Yaskawa INFORM job: kufsa_angle.JBI

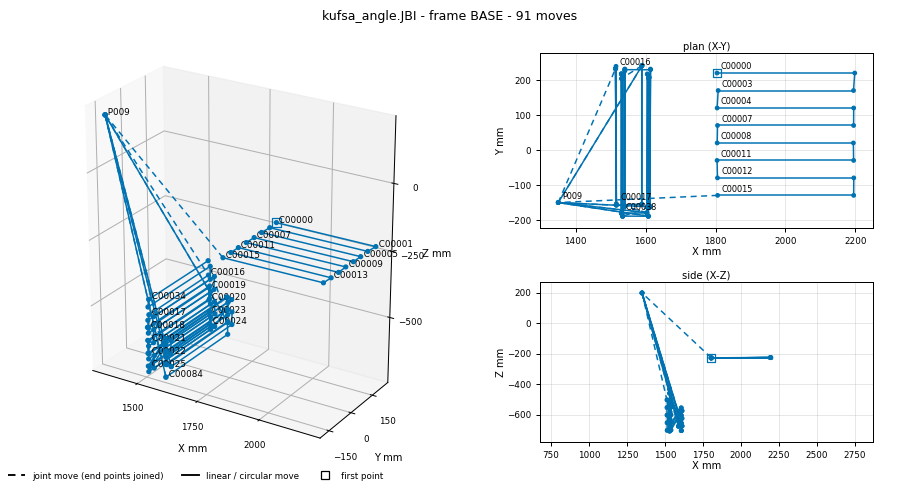
[picture p0: tool path of kufsa_angle.JBI in frame BASE, 91 of 91 moves have a stored position in this frame; points joined in program order, loops and branches not executed]
/JOB
//NAME kufsa_angle
//POS
///NPOS 86,0,86,1,0,0
///TOOL 0
///POSTYPE BASE
///RECTAN
///RCONF 0,0,0,0,0,0,0,0,0,0,0,0,0,0,0,0,0,0,0,0,0,0,0,0
C00000=1804.266,220.599,-227.332,179.0000,1.0000,1.0000
C00001=2198.370,220.599,-225.837,179.0000,1.0000,1.0000
C00002=2194.801,170.599,-225.649,179.0000,1.0000,1.0000
C00003=1807.577,170.599,-227.559,179.0000,1.0000,1.0000
C00004=1804.622,120.599,-227.769,179.0000,1.0000,1.0000
C00005=2195.335,120.599,-225.843,179.0000,1.0000,1.0000
C00006=2195.106,70.599,-225.320,179.0000,1.0000,1.0000
C00007=1805.716,70.599,-228.029,179.0000,1.0000,1.0000
C00008=1804.735,20.599,-228.045,179.0000,1.0000,1.0000
C00009=2194.418,20.599,-225.391,179.0000,1.0000,1.0000
C00010=2195.097,-29.400,-225.681,179.0000,1.0000,1.0000
C00011=1804.440,-29.400,-228.141,179.0000,1.0000,1.0000
C00012=1805.619,-79.400,-227.256,179.0000,1.0000,1.0000
C00013=2195.630,-79.400,-225.700,179.0000,1.0000,1.0000
C00014=2195.292,-129.400,-224.241,179.0000,1.0000,1.0000
C00015=1805.953,-129.400,-227.208,179.0000,1.0000,1.0000
C00016=1513.631,232.354,-503.993,179.0000,-89.9999,1.0000
C00017=1516.149,-153.231,-503.993,179.0000,-89.9999,1.0000
C00018=1516.042,-157.471,-553.993,179.0000,-89.9999,1.0000
C00019=1513.923,233.133,-553.993,179.0000,-89.9999,1.0000
C00020=1514.033,233.523,-603.993,179.0000,-89.9999,1.0000
C00021=1516.196,-156.884,-603.993,179.0000,-89.9999,1.0000
C00022=1516.145,-156.999,-653.993,179.0000,-89.9999,1.0000
C00023=1514.649,233.710,-653.993,179.0000,-89.9999,1.0000
C00024=1515.282,239.938,-703.993,179.0000,-89.9999,1.0000
C00025=1516.324,-157.007,-703.993,179.0000,-89.9999,1.0000
C00026=1588.761,-154.348,-577.217,180.0000,-45.0000,0.0000
C00027=1588.933,240.643,-577.217,180.0000,-45.0000,0.0000
C00028=1588.993,242.129,-627.217,180.0000,-45.0000,0.0000
C00029=1589.153,-155.140,-627.217,180.0000,-45.0000,0.0000
C00030=1589.056,-155.290,-677.217,180.0000,-45.0000,0.0000
C00031=1589.812,241.960,-677.217,180.0000,-45.0000,0.0000
C00032=1589.812,241.960,-677.217,180.0000,-45.0000,0.0000
C00033=1530.443,204.779,-432.522,179.0000,-89.9999,1.0000
C00034=1531.499,-175.214,-432.522,179.0000,-89.9999,1.0000
C00035=1531.405,-179.918,-459.727,179.0000,-89.9999,1.0000
C00036=1530.485,218.119,-459.727,179.0000,-89.9999,1.0000
C00037=1531.882,216.269,-509.727,179.0000,-89.9999,1.0000
C00038=1531.275,-181.949,-509.727,179.0000,-89.9999,1.0000
C00039=1531.305,-180.389,-559.727,179.0000,-89.9999,1.0000
C00040=1531.688,217.320,-559.727,179.0000,-89.9999,1.0000
C00041=1530.439,218.736,-609.727,179.0000,-89.9999,1.0000
C00042=1531.606,-180.718,-609.727,179.0000,-89.9999,1.0000
C00043=1530.852,-180.562,-659.727,179.0000,-89.9999,1.0000
C00044=1531.645,217.737,-659.727,179.0000,-89.9999,1.0000
C00045=1532.334,216.222,-709.727,179.0000,-89.9999,1.0000
C00046=1530.209,-180.083,-709.727,179.0000,-89.9999,1.0000
C00047=1603.447,-179.797,-582.950,180.0000,-45.0000,0.0000
C00048=1605.418,217.726,-582.950,180.0000,-45.0000,0.0000
C00049=1604.594,217.605,-632.950,180.0000,-45.0000,0.0000
C00050=1603.382,-179.006,-632.950,180.0000,-45.0000,0.0000
C00051=1603.382,-179.006,-632.950,180.0000,-45.0000,0.0000
C00052=1540.494,-160.372,-502.282,179.0000,-89.9999,1.0000
C00053=1540.352,230.020,-502.282,179.0000,-89.9999,1.0000
C00054=1540.533,226.582,-552.282,179.0000,-89.9999,1.0000
C00055=1540.232,-160.082,-552.282,179.0000,-89.9999,1.0000
C00056=1539.904,-161.733,-602.282,179.0000,-89.9999,1.0000
C00057=1540.218,229.622,-602.282,179.0000,-89.9999,1.0000
C00058=1540.573,232.252,-652.282,179.0000,-89.9999,1.0000
C00059=1540.340,-160.160,-652.282,179.0000,-89.9999,1.0000
C00060=1539.291,-159.918,-702.282,179.0000,-89.9999,1.0000
C00061=1540.509,230.302,-702.282,179.0000,-89.9999,1.0000
C00062=1613.808,230.041,-575.506,180.0000,-45.0000,0.0000
C00063=1612.459,-160.195,-575.506,180.0000,-45.0000,0.0000
C00064=1611.652,-164.339,-625.506,180.0000,-45.0000,0.0000
C00065=1613.824,231.968,-625.506,180.0000,-45.0000,0.0000
C00066=1613.735,230.903,-675.506,180.0000,-45.0000,0.0000
C00067=1612.429,-162.123,-675.506,180.0000,-45.0000,0.0000
C00068=1612.429,-162.123,-675.506,180.0000,-45.0000,0.0000
C00069=1534.042,-189.208,-533.001,179.0000,-89.9999,1.0000
C00070=1534.110,208.321,-533.001,179.0000,-89.9999,1.0000
C00071=1533.962,207.490,-583.001,179.0000,-89.9999,1.0000
C00072=1534.342,-189.439,-583.001,179.0000,-89.9999,1.0000
C00073=1534.609,-189.394,-633.001,179.0000,-89.9999,1.0000
C00074=1534.722,207.440,-633.001,179.0000,-89.9999,1.0000
C00075=1535.013,204.575,-683.001,179.0000,-89.9999,1.0000
C00076=1534.488,-188.796,-683.001,179.0000,-89.9999,1.0000
C00077=1607.894,-189.015,-556.224,180.0000,-45.0000,0.0000
C00078=1608.406,204.586,-556.224,180.0000,-45.0000,0.0000
C00079=1609.291,208.155,-606.224,180.0000,-45.0000,0.0000
C00080=1607.577,-189.129,-606.224,180.0000,-45.0000,0.0000
C00081=1607.618,-188.869,-656.224,180.0000,-45.0000,0.0000
C00082=1609.664,207.585,-656.224,180.0000,-45.0000,0.0000
C00083=1610.137,208.269,-706.224,180.0000,-45.0000,0.0000
C00084=1607.691,-188.817,-706.224,180.0000,-45.0000,0.0000
C00085=1607.691,-188.817,-706.224,180.0000,-45.0000,0.0000
///POSTYPE PULSE
///PULSE
EC00000=0
EC00001=0
EC00002=0
EC00003=0
EC00004=0
EC00005=0
EC00006=0
EC00007=0
EC00008=0
EC00009=0
EC00010=0
EC00011=0
EC00012=0
EC00013=0
EC00014=0
EC00015=0
EC00016=0
EC00017=0
EC00018=0
EC00019=0
EC00020=0
EC00021=0
EC00022=0
EC00023=0
EC00024=0
EC00025=0
EC00026=0
EC00027=0
EC00028=0
EC00029=0
EC00030=0
EC00031=0
EC00032=92160
EC00033=92160
EC00034=92160
EC00035=92160
EC00036=92160
EC00037=92160
EC00038=92160
EC00039=92160
EC00040=92160
EC00041=92160
EC00042=92160
EC00043=92160
EC00044=92160
EC00045=92160
EC00046=92160
EC00047=92160
EC00048=92160
EC00049=92160
EC00050=92160
EC00051=184320
EC00052=184320
EC00053=184320
EC00054=184320
EC00055=184320
EC00056=184320
EC00057=184320
EC00058=184320
EC00059=184320
EC00060=184320
EC00061=184320
EC00062=184320
EC00063=184320
EC00064=184320
EC00065=184320
EC00066=184320
EC00067=184320
EC00068=276480
EC00069=276480
EC00070=276480
EC00071=276480
EC00072=276480
EC00073=276480
EC00074=276480
EC00075=276480
EC00076=276480
EC00077=276480
EC00078=276480
EC00079=276480
EC00080=276480
EC00081=276480
EC00082=276480
EC00083=276480
EC00084=276480
EC00085=368640
///POSTYPE BASE
///RECTAN
///RCONF 1,0,0,0,0,0,0,0,0,0,0,0,0,0,0,0,0,0,0,0,0,0,0,0
P00009=1350.000,-150.000,200.000,-180.0000,-45.0000,0.0000
//INST
///DATE 2023/01/18 16:57
///ATTR SC,RW,RJ
////FRAME BASE
///GROUP1 RB1,ST1
NOP
MOVJ C00000 EC00000 VJ=15.00
CALL JOB:SPYON
MOVL C00001 EC00001 V=200.0
MOVL C00002 EC00002 V=200.0
MOVL C00003 EC00003 V=200.0
MOVL C00004 EC00004 V=200.0
MOVL C00005 EC00005 V=200.0
MOVL C00006 EC00006 V=200.0
MOVL C00007 EC00007 V=200.0
MOVL C00008 EC00008 V=200.0
MOVL C00009 EC00009 V=200.0
MOVL C00010 EC00010 V=200.0
MOVL C00011 EC00011 V=200.0
MOVL C00012 EC00012 V=200.0
MOVL C00013 EC00013 V=200.0
MOVL C00014 EC00014 V=200.0
MOVL C00015 EC00015 V=200.0
CALL JOB:SPYOF
MOVJ P009 VJ=15.00
MOVJ C00016 EC00016 VJ=15.00
CALL JOB:SPYON
MOVL C00017 EC00017 V=200.0
MOVL C00018 EC00018 V=200.0
MOVL C00019 EC00019 V=200.0
MOVL C00020 EC00020 V=200.0
MOVL C00021 EC00021 V=200.0
MOVL C00022 EC00022 V=200.0
MOVL C00023 EC00023 V=200.0
MOVL C00024 EC00024 V=200.0
MOVL C00025 EC00025 V=200.0
MOVL C00026 EC00026 V=200.0
MOVL C00027 EC00027 V=200.0
MOVL C00028 EC00028 V=200.0
MOVL C00029 EC00029 V=200.0
MOVL C00030 EC00030 V=200.0
MOVL C00031 EC00031 V=200.0
CALL JOB:SPYOF
MOVJ P009 VJ=15.00
MOVL C00032 EC00032 V=200.0
MOVJ C00033 EC00033 VJ=15.00
CALL JOB:SPYON
MOVL C00034 EC00034 V=200.0
MOVL C00035 EC00035 V=200.0
MOVL C00036 EC00036 V=200.0
MOVL C00037 EC00037 V=200.0
MOVL C00038 EC00038 V=200.0
MOVL C00039 EC00039 V=200.0
MOVL C00040 EC00040 V=200.0
MOVL C00041 EC00041 V=200.0
MOVL C00042 EC00042 V=200.0
MOVL C00043 EC00043 V=200.0
MOVL C00044 EC00044 V=200.0
MOVL C00045 EC00045 V=200.0
MOVL C00046 EC00046 V=200.0
MOVL C00047 EC00047 V=200.0
MOVL C00048 EC00048 V=200.0
MOVL C00049 EC00049 V=200.0
MOVL C00050 EC00050 V=200.0
CALL JOB:SPYOF
MOVJ P009 VJ=15.00
MOVL C00051 EC00051 V=200.0
MOVJ C00052 EC00052 VJ=15.00
CALL JOB:SPYON
MOVL C00053 EC00053 V=200.0
MOVL C00054 EC00054 V=200.0
MOVL C00055 EC00055 V=200.0
MOVL C00056 EC00056 V=200.0
MOVL C00057 EC00057 V=200.0
MOVL C00058 EC00058 V=200.0
MOVL C00059 EC00059 V=200.0
MOVL C00060 EC00060 V=200.0
MOVL C00061 EC00061 V=200.0
MOVL C00062 EC00062 V=200.0
MOVL C00063 EC00063 V=200.0
MOVL C00064 EC00064 V=200.0
MOVL C00065 EC00065 V=200.0
MOVL C00066 EC00066 V=200.0
MOVL C00067 EC00067 V=200.0
CALL JOB:SPYOF
MOVJ P009 VJ=15.00
MOVL C00068 EC00068 V=200.0
MOVJ C00069 EC00069 VJ=15.00
CALL JOB:SPYON
MOVL C00070 EC00070 V=200.0
MOVL C00071 EC00071 V=200.0
MOVL C00072 EC00072 V=200.0
MOVL C00073 EC00073 V=200.0
MOVL C00074 EC00074 V=200.0
MOVL C00075 EC00075 V=200.0
MOVL C00076 EC00076 V=200.0
MOVL C00077 EC00077 V=200.0
MOVL C00078 EC00078 V=200.0
MOVL C00079 EC00079 V=200.0
MOVL C00080 EC00080 V=200.0
MOVL C00081 EC00081 V=200.0
MOVL C00082 EC00082 V=200.0
MOVL C00083 EC00083 V=200.0
MOVL C00084 EC00084 V=200.0
CALL JOB:SPYOF
MOVJ P009 VJ=15.00
MOVL C00085 EC00085 V=200.0
END
